GLOBALCONSTANTS logiBUS_2_CAN_DI (* logiBUS_DI constants *)
  (* Standard: 61499-1; Description: Copyright (c) 2024 HR Agrartechnik GmbH This program and the accompanying materials are made available under the terms of the Eclipse Public License 2.0 which is available at https://www.eclipse.org/legal/epl-2.0/ SPDX-License-Identifier: EPL-2.0 *)
  (* Version 1.0, 2024-01-25, Franz Höpfinger, HR Agrartechnik GmbH *)
  PACKAGE logiBUS::io::DI_CAN;
  VAR_GLOBAL CONSTANT
    Input_CI1 : logiBUS::io::DI_CAN::logiBUS_2_CAN_DI_S := (Pin := 1);
    Input_CI2 : logiBUS::io::DI_CAN::logiBUS_2_CAN_DI_S := (Pin := 2);
    Invalid : logiBUS::io::DI_CAN::logiBUS_2_CAN_DI_S := (Pin := 255);
  END_VAR
END_GLOBALCONSTANTS
